FUNCTION_BLOCK FB_SpindleZ EXTENDS FB_PackML_BaseModule
VAR
    // Sub module definitions here

    // List of sub modules
    ipSubModules_Init : ARRAY[1..Parameters_PackML_Base.MAX_NO_OF_SUBMODULES] OF I_PackML_BaseModule := [];

    // Component definitions here
    Axis   : FB_Component_BasicAxis := (Name := 'Axis');
    Sensor : FB_DigitalSensor       := (Name := 'Sensor');

    //Alarms for this module
    SpindleAlarms : ARRAY[1..SPINDLE_ALARM_COUNT] OF FB_TcAlarm;

    //Data for recipe


    (*Parameters from PackTags for module
    //_Param  : ARRAY[1..10] OF ST_Descriptor2;*)
    _Report : ARRAY[1..10] OF ST_Descriptor2;

    //HMI Control for EM
    fbControlSourceHMI : FB_ControlSource_HMI;
END_VAR

VAR CONSTANT
    //reports 
    FAULT : INT := 1;

    //Alarms
    SPINDLE_ALARM_COUNT : INT := 5;
END_VAR

//Simulation variables for messaging
VAR
    ErrorInput : BOOL;
    WarnInput  : BOOL;
    InfoInput  : BOOL;
END_VAR

METHOD PROTECTED CreateEvents
VAR_INPUT
END_VAR
// Add your event creation here
F_CreateAllEventsInClass(Alarms     := SpindleAlarms,
                         ClassSize  := SIZEOF(TC_EVENTS.Spindle),
                         pInitEvent := ADR(TC_EVENTS.Spindle.InitReferenceEvent),
                         Prefix     := Name);

// Super call to base
SUPER^.CreateEvents();
END_METHOD

METHOD CyclicLogic
VAR_INPUT
END_VAR
IF NOT _InitComplete THEN
    _InitComplete := Initialize();
    RETURN;
END_IF

SUPER^.CyclicLogic();

//HMI control for EM
fbControlSourceHMI.CyclicLogic();

//Set the current alarm severity for this module
_CurrentAlarmSeverity := F_GetMaxSeverityRaised(Alarms := SpindleAlarms, CurrentSeverity := _CurrentAlarmSeverity);
IF _CurrentAlarmSeverity >= TcEventSeverity.Error THEN
    ChangeState(E_PMLCommand.ePMLCommand_Abort);
END_IF
END_METHOD

//! @summary Basic module initialization logic
METHOD PROTECTED Initialize : BOOL;
VAR
    i                        : UDINT;
    varInfo                  : __SYSTEM.VAR_INFO;
    AllSubUnitsInitialized   : BOOL := TRUE;
    AllComponentsInitialized : BOOL := TRUE;
END_VAR

//! @description This method is called by <c>CyclicLogic()</c> as required
Initialize := FALSE;
CASE DescendantSequenceState OF
    0:
		RegisterComponent(Axis);
		RegisterComponent(Sensor);
        _LogModeChanges         := TRUE;
        _LogStateChanges        := TRUE;
        DescendantSequenceState := DescendantSequenceState + 10;
    10:
        //Setup Custom modes here

        (*CustomModes(eMode                          :=,
                    sName                          :=,
                    bDisableClearing               :=,
                    bDisableStarting               :=,
                    bDisableSuspended              :=,
                    bDisableStopping               :=,
                    bDisableAborting               :=,
                    bDisableHolding                :=,
                    bDisableHeld                   :=,
                    bDisableUnholding              :=,
                    bDisableSuspending             :=,
                    bDisableUnsuspending           :=,
                    bDisableResetting              :=,
                    bDisableIdle                   :=,
                    bDisableCompleting             :=,
                    bDisableComplete               :=,
                    bEnableUnitModeChangeStopped   :=,
                    bEnableUnitModeChangeIdle      :=,
                    bEnableUnitModeChangeSuspended :=,
                    bEnableUnitModeChangeExecute   :=,
                    bEnableUnitModeChangeAborted   :=,
                    bEnableUnitModeChangeHeld      :=,
                    bEnableUnitModeChangeComplete  :=,
                    bError                         =>,
                    nErrorId                       =>);*)
        DescendantSequenceState := DescendantSequenceState + 10;
    20:
        //Copy Mode names
        FOR i := 1 TO 3 DO
            ModeNames[i] := F_UnitModeToString(UDINT_TO_DINT(i));
        END_FOR

 
		RegisterExternalController(Controller := fbControlSourceHMI);
		fbControlSourceHMI.CyclicLogic();
		
		//Set the Parent Response here
		_ParentFaultResponseDefinitions[TcEventSeverity.Error] := E_AlarmResponse.Hold_Immediate;
        DescendantSequenceState := DescendantSequenceState + 10;
    30:
        //Call the Super
        IF SUPER^.Initialize() THEN
            DescendantSequenceState := DescendantSequenceState + 10;
        END_IF
    40:
        Initialize := TRUE;
END_CASE
END_METHOD

METHOD RaiseAlarm2Args
VAR_IN_OUT
    Alarm : FB_TcAlarm; //Alarm to be raised
END_VAR

VAR_INPUT
    String_1 : STRING; //First String Parameter (The Name of this component will be applied first automatically)
    String_2 : STRING; //Second String Parameter
END_VAR
F_RaiseAlarmWithStringParameters(Alarm    := Alarm,
                                 String_1 := Name,
                                 String_2 := String_1,
                                 String_3 := String_2);
END_METHOD

END_FUNCTION_BLOCK

(* stored: Version 1.1.0.1
   POU FB_SpindleZ: Id {93b6d370-9060-40d7-8101-95f7e4ba6901}, SpecialFunc None
   Folder I_CyclicFB: Id {50b2b73b-a7e6-449c-8083-d6eb4b73f60c}
   Folder Methods: Id {1fe8be3a-f7d7-42ae-b885-2501b85559e1}
   Method CreateEvents: Id {99ddd031-78aa-46a7-b2f9-f0b68a19d02e}
   Method CyclicLogic: Id {ea09e275-dd4c-4ec1-a323-7e0cfd7e21cd}
   Method Initialize: Id {59d1fe7d-28ec-4cbf-a3ef-81f06735b3ba}
   Method RaiseAlarm2Args: Id {7b5fcd4f-47a7-4be3-b737-1f985fad3866} *)
